(* IEC 61131-3 sources: RAG_PLC/data/result/test/056, 2 files *)

(* ---- wrapped.st ---- *)
(* =========================================================
   Generated by PLC-Eval Benchmark Wrapper
   ========================================================= *)

FUNCTION_BLOCK LLM_Wrapper_FB
VAR_INPUT
    STR : STRING;
END_VAR

VAR_OUTPUT
    STR_TO_DW : DWORD;
END_VAR

VAR
    TEMP : STRING[10];
    I : INT;
    CHAR_VAL : BYTE;
    RESULT : DWORD;
END_VAR

TEMP := STR;
RESULT := DWORD#0;

FOR I := 1 TO LEN(TEMP) DO
    CHAR_VAL := BYTE(TEMP[I]);
    IF CHAR_VAL >= BYTE('0') AND CHAR_VAL <= BYTE('9') THEN
        RESULT := RESULT * DWORD#10 + DWORD(CHAR_VAL - BYTE('0'));
    ELSIF CHAR_VAL >= BYTE('A') AND CHAR_VAL <= BYTE('F') THEN
        RESULT := RESULT * DWORD#16 + DWORD(CHAR_VAL - BYTE('A') + 10);
    ELSIF CHAR_VAL >= BYTE('a') AND CHAR_VAL <= BYTE('f') THEN
        RESULT := RESULT * DWORD#16 + DWORD(CHAR_VAL - BYTE('a') + 10);
    END_IF;
END_FOR;

STR_TO_DW := RESULT;
END_FUNCTION_BLOCK

PROGRAM Auto_Proxy_Prg
  VAR
    instance : LLM_Wrapper_FB;
  END_VAR

  instance();
END_PROGRAM

CONFIGURATION Config0
  RESOURCE Res0 ON PLC
    TASK TaskMain(INTERVAL := T#20ms, PRIORITY := 0);
    PROGRAM Inst0 WITH TaskMain : Auto_Proxy_Prg;
  END_RESOURCE
END_CONFIGURATION

(* ---- raw_code.st ---- *)
VAR_INPUT
    STR : STRING;
END_VAR

VAR_OUTPUT
    STR_TO_DW : DWORD;
END_VAR

VAR
    TEMP : STRING[10];
    I : INT;
    CHAR_VAL : BYTE;
    RESULT : DWORD;
END_VAR

TEMP := STR;
RESULT := DWORD#0;

FOR I := 1 TO LEN(TEMP) DO
    CHAR_VAL := BYTE(TEMP[I]);
    IF CHAR_VAL >= BYTE('0') AND CHAR_VAL <= BYTE('9') THEN
        RESULT := RESULT * DWORD#10 + DWORD(CHAR_VAL - BYTE('0'));
    ELSIF CHAR_VAL >= BYTE('A') AND CHAR_VAL <= BYTE('F') THEN
        RESULT := RESULT * DWORD#16 + DWORD(CHAR_VAL - BYTE('A') + 10);
    ELSIF CHAR_VAL >= BYTE('a') AND CHAR_VAL <= BYTE('f') THEN
        RESULT := RESULT * DWORD#16 + DWORD(CHAR_VAL - BYTE('a') + 10);
    END_IF;
END_FOR;

STR_TO_DW := RESULT;
